PROGRAM P_Demo_FB_DMXGetProductDetailIdList
VAR
    fbGetProdDetails  : FB_DMXGetProductDetailIdList; // 读产品类别列表
    stDmxCmdBuffer    : ST_DMXCommandBuffer;          // 与通讯 FB 共用
    wTargetManufId    : WORD := 16#4241;              // 目标灯具厂商 ID
    dwTargetDeviceId  : DWORD := 16#12131415;         // 目标灯具设备 ID
    byTargetPort      : BYTE := 0;                    // 根设备通道 0
    bDoRead           : BOOL := FALSE;                // 在线给一次上升沿触发
    bBusy             : BOOL;
    bError            : BOOL;
    udiErrId          : UDINT;
    arrProdDetails    : ARRAY [1..6] OF E_DMXProductDetail;  // 产品类别（最多 6）
END_VAR

// ============================================================
// Tc2_DMX.FB_DMXGetProductDetailIdList 演示程序
// ============================================================
// 场景：按功能给灯具自动分组：读出每台设备产品类别，把调光器/染色灯/烟机等分别归类供分组控制。
// 价值：把设备功能类别从设备直接读出，可实现自动化设备分类，免去人工按型号归类。
// 验证：给 bDoRead 一次上升沿 -> bBusy 短暂 TRUE -> 回 FALSE 后 arrProdDetails[1..6] 含设备产品类别枚举值。
// 验证步骤：
//   1. 右键 PLC 项目下 POUs 文件夹 → Add → Existing Item → 选本 .TcPOU 文件
//   2. 引用 Tc2_DMX；同项目里放一个 FB_EL6851CommunicationEx 实例并共用 stDmxCmdBuffer（非 CycleMode）
//   3. 编译 → 登录 → 运行；按上方『验证』行在线给上升沿观察
// ============================================================

fbGetProdDetails(
    bStart                     := bDoRead,
    wDestinationManufacturerId := wTargetManufId,
    dwDestinationDeviceId      := dwTargetDeviceId,
    byPortId                   := byTargetPort,
    dwOptions                  := 0,
    stCommandBuffer            := stDmxCmdBuffer,
    bBusy                      => bBusy,
    bError                     => bError,
    udiErrorId                 => udiErrId,
    arrProductDetails          => arrProdDetails
);

END_PROGRAM

(* stored: Version 1.1.0.1, ProductVersion 3.1.4024.5
   POU P_Demo_FB_DMXGetProductDetailIdList: Id {13f69729-e665-5f8b-a566-95531eb970e7}, SpecialFunc None *)
